(* PLC project Unnamed, Unknown Unnamed 1 *)
(* stored: creationDateTime 2022-10-16T10:53:06, modificationDateTime 2022-10-16T17:55:15 *)

PROGRAM Actuators
  VAR
    PON00 AT %IX0.0 : BOOL;
    PON01 AT %IX0.1 : BOOL;
    PON02 AT %IX0.2 : BOOL;
    PON03 AT %IX0.3 : BOOL;
    PON04 AT %IX0.4 : BOOL;
    PON05 AT %IX0.5 : BOOL;
    PON06 AT %IX0.6 : BOOL;
    PON07 AT %IX0.7 : BOOL;
    POF00 AT %IX1.0 : BOOL;
    POF01 AT %IX1.1 : BOOL;
    POF02 AT %IX1.2 : BOOL;
    POF03 AT %IX1.3 : BOOL;
    POF04 AT %IX1.4 : BOOL;
    POF05 AT %IX1.5 : BOOL;
    POF06 AT %IX1.6 : BOOL;
    POF07 AT %IX1.7 : BOOL;
    LED00 AT %QX0.0 : BOOL;
    LED01 AT %QX0.1 : BOOL;
    LED02 AT %QX0.2 : BOOL;
    LED03 AT %QX0.3 : BOOL;
    LED04 AT %QX0.4 : BOOL;
    LED05 AT %QX0.5 : BOOL;
    LED06 AT %QX0.6 : BOOL;
    LED07 AT %QX0.7 : BOOL;
  END_VAR

(* LD diagram, written out as Structured Text *)
LED00 := (LED00 OR PON00) AND NOT POF00;
LED01 := (LED01 OR PON01) AND NOT POF01;
LED02 := (LED02 OR PON02) AND NOT POF02;
LED03 := (LED03 OR PON03) AND NOT POF03;
LED04 := (LED04 OR PON04) AND NOT POF04;
LED05 := (LED05 OR PON05) AND NOT POF05;
LED06 := (LED06 OR PON06) AND NOT POF06;
LED07 := (LED07 OR PON07) AND NOT POF07;
END_PROGRAM

CONFIGURATION Config0
  RESOURCE Res0 ON PLC
    TASK task0(INTERVAL := T#20ms, PRIORITY := 0);
    PROGRAM instance0 WITH task0 : Actuators;
  END_RESOURCE
END_CONFIGURATION
